{attribute 'call_after_init'}
FUNCTION_BLOCK FB_AssertTrueFalse_Test EXTENDS TcUnit.FB_TestSuite IMPLEMENTS TcUnit.I_RunnableTestSuite
VAR
    Assert : TcUnit.FB_Assert;
END_VAR

METHOD PRIVATE AssertThatINTsAreEqual
VAR
    a : INT := -33;
    b : INT := -44;
END_VAR
TEST('AssertThatINTsAreEqual');

Assert.AssertFalse(Condition := (a <> b),
                   Message := 'INTs are equal');
END_METHOD

METHOD PRIVATE AssertThatINTsAreNotEqual
VAR
    a : INT := -33;
    b : INT := -44;
END_VAR
TEST('AssertThatINTsAreNotEqual');

Assert.AssertFalse(Condition := (a = b),
                   Message := 'INTs are equal');
END_METHOD

METHOD PRIVATE AssertThatWORDsAreEqual
VAR
    a : WORD := 16#ABCD;
    b : WORD := 16#0123;
END_VAR
TEST('AssertThatWORDsAreEqual');

Assert.AssertTrue(Condition := (a = b),
                  Message := 'WORDs are not equal');
END_METHOD

METHOD PRIVATE AssertThatWORDsAreNotEqual
VAR
    a : WORD := 16#ABCD;
    b : WORD := 16#0123;
END_VAR
TEST('AssertThatWORDsAreNotEqual');

Assert.AssertTrue(Condition := (a <> b),
                  Message := 'WORDs are equal');
END_METHOD

METHOD FB_init : BOOL
VAR_INPUT
	bInitRetains : BOOL; // if TRUE, the retain variables are initialized (warm start / cold start)
	bInCopyCode : BOOL;  // if TRUE, the instance afterwards gets moved into the copy code (online change)
END_VAR
SUPER^.RegisterTestSuite(THIS^);
END_METHOD

METHOD RunTests : TCUNIT.E_TestSuiteRunState
AssertThatINTsAreEqual();
AssertThatINTsAreNotEqual();
AssertThatWORDsAreEqual();
AssertThatWORDsAreNotEqual();

RunTests := TCUNIT.E_TestSuiteRunState.FINISHED;
END_METHOD

END_FUNCTION_BLOCK

(* stored: Version 1.1.0.1, ProductVersion 3.1.4022.12
   POU FB_AssertTrueFalse_Test: Id {4a344c15-007d-4e24-b34e-25e793163fe6}, SpecialFunc None
   Method AssertThatINTsAreEqual: Id {e329edff-158b-47b8-b448-4482e312fc51}
   Method AssertThatINTsAreNotEqual: Id {e9713416-6687-4536-b3eb-d0e312881039}
   Method AssertThatWORDsAreEqual: Id {cb8a8728-6b7f-485b-9255-e9e2c3d7b1b4}
   Method AssertThatWORDsAreNotEqual: Id {7f2e9dc0-aaa1-4524-9220-4e31b7d76d84}
   Method FB_init: Id {d9c8d1d8-437d-4506-86dc-1943db55bc24}
   Method RunTests: Id {f30a7ae9-e875-48f2-9a5e-ace6bb6be399} *)
